FUNCTION_BLOCK PID3_Manager (* Composite Function Block Type *)
  (* Standard: 61499-2 *)
  (* Version 0.0, 12/17/2025, SESA313294, Schneider Electric, template *)
  PACKAGE SE.Nereda;
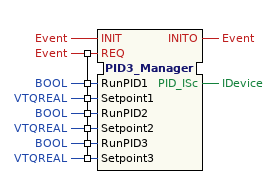
  EVENT_INPUT
    INIT; (* Initialization *)
    REQ WITH RunPID1, Setpoint1, RunPID2, Setpoint2, RunPID3, Setpoint3; (* Normal Execution Request *)
  END_EVENT
  EVENT_OUTPUT
    INITO; (* Initialization Confirmation *)
  END_EVENT
  VAR_INPUT
    RunPID1 : BOOL;
    Setpoint1 : VTQREAL;
    RunPID2 : BOOL;
    Setpoint2 : VTQREAL;
    RunPID3 : BOOL;
    Setpoint3 : VTQREAL;
  END_VAR
  PLUGS
    PID_ISc : IDevice;
  END_PLUGS
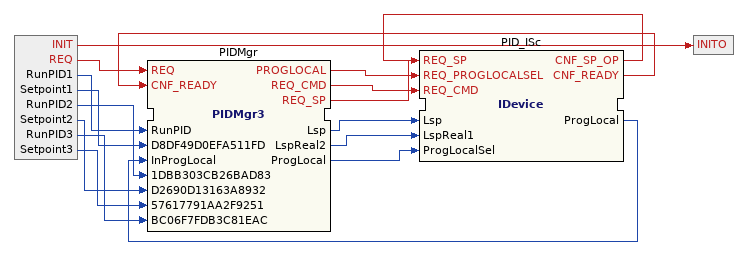
  FBS
    PIDMgr : PIDMgr3;
  END_FBS
  EVENT_CONNECTIONS
    PID_ISc.CNF_SP_OP TO PID_ISc.REQ_SP;
    REQ TO PIDMgr.REQ;
    PID_ISc.CNF_READY TO PIDMgr.CNF_READY;
    PIDMgr.PROGLOCAL TO PID_ISc.REQ_PROGLOCALSEL;
    PIDMgr.REQ_CMD TO PID_ISc.REQ_CMD;
    INIT TO INITO;
    PIDMgr.REQ_SP TO PID_ISc.REQ_SP;
  END_CONNECTIONS
  DATA_CONNECTIONS
    RunPID1 TO PIDMgr.RunPID;
    Setpoint1 TO PIDMgr.D8DF49D0EFA511FD;
    PIDMgr.Lsp TO PID_ISc.Lsp;
    PIDMgr.LspReal2 TO PID_ISc.LspReal1;
    PIDMgr.ProgLocal TO PID_ISc.ProgLocalSel;
    PID_ISc.ProgLocal TO PIDMgr.InProgLocal;
    RunPID2 TO PIDMgr.1DBB303CB26BAD83;
    Setpoint2 TO PIDMgr.D2690D13163A8932;
    Setpoint3 TO PIDMgr.57617791AA2F9251;
    RunPID3 TO PIDMgr.BC06F7FDB3C81EAC;
  END_CONNECTIONS
END_FUNCTION_BLOCK
